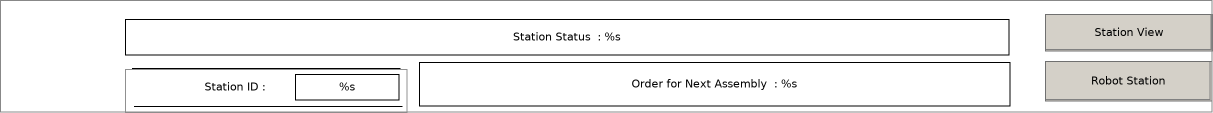
VISUALIZATION Visualization  // 1213x113
    Rectangle (125,19 884x36), "Station Status : %s", text variable: Visualaisation_Control.mxStationStatus
    GroupBox (125,61 282x52)
        Line (6,458) (274,458)
        Line (7,7) (275,7)
        Label (35,11 150x30), "Station ID :"
        Rectangle (170,13 104x26), "%s", text variable: GVL.mwStationID
        Line (9,45) (277,45)
    Button (1045,61 167x40), "Robot Station"
        OnMouseClick: change screen: RobotStation
    Rectangle (419,62 591x44), "Order for Next Assembly : %s", text variable: GVL.qsOrderFornextAssembly
    Button (1045,14 168x37), "Station View"
        OnMouseClick: change screen: Station
END_VISUALIZATION

(* stored: Version 1.1.0.1, ProductVersion 3.1.4024.12
   Visu Visualization: Id {08c1f753-3e44-4c26-b458-35ef78727ab8} *)
